// TIA Portal V20 export
TYPE "typeSafetyDoorBox"
// stored: Access Published, IsFailsafeCompliant true, Namespace Safety
   STRUCT
      SI1_Lock_PB : Bool;
      SI2_Unlock_PB : Bool;
      SI3_Reset_PB : Bool;
      SO1_Lock_PL : Bool;
      SO2_Unlock_PL : Bool;
      SO3_Reset_PL : Bool;
   END_STRUCT;
END_TYPE
